% RSLogix 500 project UNTITLED_BAK014.RSS, saved by version 8.10.00.18 %
PROJECT "UNTITLED"    % processor: MicroLogix 1200 %

PROGRAM FILES
  LAD 2   4 rungs

DATA FILES
  O0 OUTPUT  4 elements
  I1 INPUT  4 elements
  S2 STATUS  66 elements
  B3 BINARY  1 elements
  T4 TIMER  1 elements
  C5 COUNTER  1 elements
  R6 CONTROL  1 elements
  N7 INTEGER  1 elements

LADDER 2
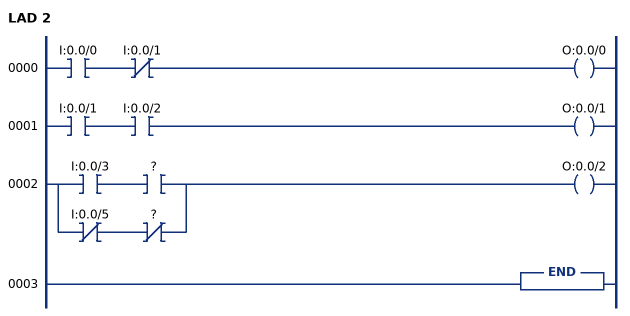
% Rung: 0 %
SOR XIC I:0.0/0 XIO I:0.0/1 OTE O:0.0/0 EOR
% Rung: 1 %
SOR XIC I:0.0/1 XIC I:0.0/2 OTE O:0.0/1 EOR
% Rung: 2 %  % edit flag set %
SOR BST XIC I:0.0/3 XIC ? NXB XIO I:0.0/5 XIO ? BND OTE O:0.0/2 EOR
% Rung: 3 %
SOR END EOR
